Staubli VAL3: oHeaterTask.pgx

program oHeaterTask(num nDuration (dimensions=1))
// Heater
begin
  dioSet(oHeater,1)
  delay(nDuration)
  dioSet(oHeater,0)
end
